// TIA Portal V20 export
TYPE "typeEm6MonitoringJobInterface"
// stored: Access Published, Namespace Unit1
   STRUCT
      busyVisionInspection { ExternalWritable := 'False'} : Bool;
      doneVisionInspection { ExternalWritable := 'False'} : Bool;
      busyQrRead { ExternalWritable := 'False'} : Bool;
      doneQrRead { ExternalWritable := 'False'} : Bool;
   END_STRUCT;
END_TYPE
